(*
	Function Block which performs a level control using a DOL pump and a high level switch
*)
{attribute 'OPC.UA.DA.StructuredType' := '1'}
FUNCTION_BLOCK FB_ControlLoop_DissOx EXTENDS FB_BaseDevice
VAR_IN_OUT
	fbInjector: 			FB_OxygenInjector;
	fbSensorDissOx: 		FB_Sensor_AtlasDO;
	nSetPoint:				REAL;
END_VAR


VAR PERSISTENT
	tDebounce: TIME := T#1M; 
END_VAR

VAR
	bFirstRun: BOOL := TRUE;
	eSMState: (WAIT, DOSE_ON, DOSE_OFF, TURNING_OFF);
	fbTON_Debouce: TON := (PT := tDebounce, IN := FALSE);

END_VAR

IF bFirstRun THEN
	
	bFirstRun := FALSE;
END_IF


IF GVL.bAutoUpdateDeviceState THEN
	eState := eStateTarget;	
END_IF


IF eMode = E_DeviceMode.MANUAL OR eStateTarget = E_DeviceState.ON THEN
	bEnable := TRUE;
	fbInjector.enable();
END_IF

IF bEnable AND (eStateTarget = E_DeviceState.ON) AND (eSMState <> DOSE_ON) THEN
		eSMState := DOSE_OFF;
		fbInjector.enable();
END_IF


IF (bEnable = FALSE) OR (eStateTarget = E_DeviceState.OFF) THEN
		eSMState := TURNING_OFF;
		fbInjector.disable();
END_IF


IF bEnable THEN
	CASE eSMState OF
		WAIT:
			// Do nothing
			eState := E_DeviceState.OFF;
			
			
		DOSE_OFF:
			fbTON_Debouce(PT := tDebounce, IN := TRUE);
			eState := E_DeviceState.ON;
			fbInjector.setCommand(StateTarget := E_DeviceState.OFF);
			IF (fbSensorDissOx.getValue() < nSetPoint)  AND (fbTON_Debouce.Q) THEN
				eSMState := DOSE_ON;
			END_IF
			
		DOSE_ON:
			fbTON_Debouce(IN := FALSE);
			eState := E_DeviceState.ON;
			fbInjector.setCommand(StateTarget := E_DeviceState.ON);
			IF (fbSensorDissOx.getValue() > nSetPoint)THEN
				eSMState := DOSE_OFF;
			END_IF
			
		TURNING_OFF:
			eState := E_DeviceState.TURNING_OFF;
			fbInjector.setCommand(StateTarget := E_DeviceState.OFF);
			eSMState := WAIT;
			
	END_CASE
END_IF

METHOD setState : BOOL
VAR_INPUT
	state : E_DeviceState;
END_VAR

eState := state;
END_METHOD

END_FUNCTION_BLOCK

(* stored: Version 1.1.0.1, ProductVersion 3.1.4024.12
   POU FB_ControlLoop_DissOx: Id {82094251-7bb9-4cce-aa77-5198aa8377e5}, SpecialFunc None
   Method setState: Id {5836fcd8-d635-419e-aa2c-5f02430854b9} *)
